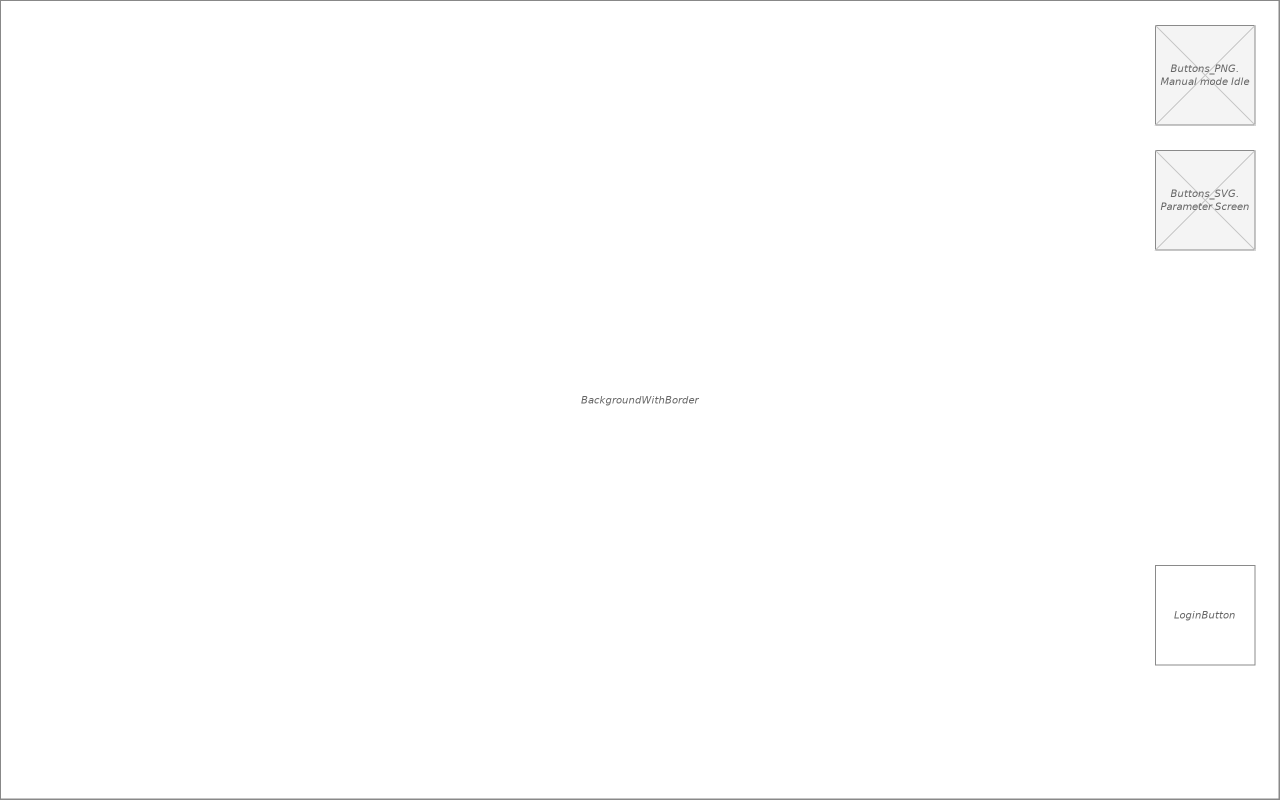
VISUALIZATION BaseScreen  // 1280x800
    Frame (0,0 1280x800)
        shows BackgroundWithBorder()
    Frame (1155,565 100x100), invisible if: GVL_HMI.fbHMIControl.bHideBorders
        shows LoginButton()
    Image (1155,150 100x100), invisible if: GVL_HMI.fbHMIControl.bHideBorders, image: Buttons_SVG.Parameter Screen
        OnMouseDown: toggle GVL_HMI.bCmdParameter
    Image (1155,25 100x100), invisible if: GVL_HMI.fbHMIControl.bHideBorders, image: Buttons_PNG.Manual mode Idle
        OnMouseDown: toggle GVL_HMI.bCmdManual
END_VISUALIZATION

(* stored: Version 1.1.0.1, ProductVersion 3.1.4024.11
   Visu BaseScreen: Id {4947af5d-5d50-4f16-ab4a-243dcb1607d8} *)
